(* LS Electric XG5000 project: V2H *)
(* PLC NewPLC *)
(* module base 0 slot 0: Input/Output Module:XEC-DR64H (DC 24V INPUT/RELAY OUTPUT, 64points) *)
(* module base 0 slot 1: Analog Input Module:XBF-AD04A (Volt/Current, 4-CH) *)
(* module base 0 slot 2: Analog IO Module:XBF-AH04A (I/O, 2/2 CH) *)
VAR_GLOBAL
    _01_CH0_ACT AT %UX0.1.16 : BOOL; (* Analog Input Module: CH0 Active *)
    _01_CH0_DATA AT %UW0.1.2 : WORD; (* Analog Input Module: CH0 Output *)
    _01_CH1_ACT AT %UX0.1.17 : BOOL; (* Analog Input Module: CH1 Active *)
    _01_CH1_DATA AT %UW0.1.3 : WORD; (* Analog Input Module: CH1 Output *)
    _01_CH2_ACT AT %UX0.1.18 : BOOL; (* Analog Input Module: CH2 Active *)
    _01_CH2_DATA AT %UW0.1.4 : WORD; (* Analog Input Module: CH2 Output *)
    _02_DA0_ACT AT %UX0.2.18 : BOOL; (* Analog IO Module: Output CH0 Active *)
    _02_DA0_OUTEN AT %UX0.2.96 : BOOL; (* Analog IO Module: Output CH0 Status Setting *)
    _02_DA1_DATA AT %UW0.2.8 : WORD; (* Analog IO Module: Output CH1 DATA *)
END_VAR

PROGRAM NewProgram_Copy (* task: Scan Program *)
VAR
    aa : REAL;
    AAAA : WORD;
    aaaaaaaaaaaaaaa : REAL;
    acCONTROL AT %IX0.0.0 : BOOL;
    ACTRANS : BOOL;
    ADD1 : WORD;
    ADD2 : WORD;
    AUTO AT %MX1 : BOOL;
    autoinhibit : BOOL;
    BLOCK : UINT;
    chillerready : BOOL;
    COMPRESSOR : BOOL;
    CONACTOR100 AT %IX0.0.21 : BOOL;
    CONTACTOR10 AT %IX0.0.3 : BOOL;
    CONTACTOR20 AT %IX0.0.4 : BOOL;
    CONTACTOR30 AT %IX0.0.8 : BOOL;
    CONTACTOR40 AT %IX0.0.9 : BOOL;
    CONTACTOR50 AT %IX0.0.10 : BOOL;
    CRITICALPRESSURE : BOOL;
    damperon : BOOL;
    damperramp : BOOL;
    DAMPERREF : WORD;
    DCPOWERK : BOOL;
    ddddddd : BOOL;
    DIRTYFILTER : BOOL;
    disk11kman : BOOL;
    disk1kman : BOOL;
    DIV11 : WORD;
    DIV12 : INT;
    DIV124 : INT;
    DIV2 : WORD;
    DIV21 : WORD;
    DIV22 : WORD;
    DIV23 : WORD;
    DIV32 : INT;
    DIV33 : INT;
    DP1SUBP1MACHIN : WORD;
    DP1SUBP1MACHIN2 : WORD;
    DP1SUBP1MACHININT : INT;
    DP2INT : INT;
    DP2RATE : INT;
    DPINT : INT;
    DPMUL : WORD;
    DPSUBZERO : INT;
    drive11kman : BOOL;
    DRIVE11KW AT %QX0.0.10 : BOOL;
    DRIVE75KW AT %QX0.0.9 : BOOL;
    DRIVEK1 AT %MX90 : BOOL;
    DRIVEK2 AT %MX91 : BOOL;
    DRIVEK3 : BOOL;
    DRIVEK4 : BOOL;
    DRIVEK5 : BOOL;
    DRIVEK6 : BOOL;
    DRIVEPUMP AT %MX92 : BOOL;
    dvi2 : DWORD;
    E1 : INT;
    E11 : REAL;
    E1REAL : REAL;
    E2 : WORD;
    EE : WORD;
    EE1 : WORD;
    EE2 : WORD;
    EMERGENCY AT %IX0.0.23 : BOOL;
    ERR : BOOL;
    ET : TIME;
    ET70 : TIME;
    fanon : BOOL;
    FANREFSCALE : WORD;
    FANRUN : BOOL;
    filterdisk : BOOL;
    filterjaroob : BOOL;
    FILTERMEDIA : BOOL;
    FILTERRUN : BOOL;
    FR1 AT %IX0.0.14 : BOOL;
    FR2 AT %IX0.0.15 : BOOL;
    FR3 AT %IX0.0.16 : BOOL;
    FR4 AT %IX0.0.17 : BOOL;
    FR5 AT %IX0.0.18 : BOOL;
    FR6 AT %IX0.0.19 : BOOL;
    GEARBOXK5 AT %QX0.0.5 : BOOL;
    gearboxman : BOOL;
    HIGHLIMDP : WORD;
    hihelimdpint : INT;
    HIMIDITYSCAL2 : WORD;
    HUMID2 : WORD;
    HUMID3 : WORD;
    HUMID4 : BOOL;
    HUMID5 : BOOL;
    HUMIDHIVALUE1 : WORD;
    HUMIDITIERR1 : WORD;
    HUMIDITYOUTSCAL : WORD;
    HUMIDLOWLIM1 : WORD;
    HUMIDNO1 : BOOL;
    HUMIDON : BOOL;
    hummidd : WORD;
    IN1 : SINT;
    IN10 : WORD;
    incin : WORD;
    inhumreal : REAL;
    inhumreal1 : REAL;
    inrealhuscale : REAL;
    inrealhuscale1 : REAL;
    INST : TON;
    INST1 : TON;
    INST10 : PIDRUN;
    INST11 : PIDRUN;
    INST12 : TON_UINT;
    INST13 : TON_UINT;
    INST14 : TON;
    INST15 : TON;
    INST16 : TON;
    INST17 : TON;
    INST18 : TON;
    INST19 : TON;
    INST2 : TON;
    INST20 : TON;
    INST21 : TON;
    INST22 : TON;
    INST23 : TON;
    INST24 : TON;
    INST25 : TON;
    INST26 : CTU_INT;
    INST27 : TON;
    INST28 : TON;
    INST29 : CTU_INT;
    INST3 : TON;
    INST30 : TON;
    INST31 : TON;
    INST32 : TON;
    INST33 : TON;
    INST34 : TON;
    INST35 : TON;
    INST36 : TON;
    INST37 : CTU_INT;
    INST38 : CTU_INT;
    INST39 : TON;
    INST4 : TON;
    INST40 : TON_UINT;
    INST41 : TON_UINT;
    INST42 : TON_UINT;
    INST43 : TON_UINT;
    INST44 : TON_UINT;
    INST45 : TON_UINT;
    INST46 : TON_UINT;
    INST47 : TMR;
    INST48 : TON_UINT;
    INST49 : TON_UINT;
    INST5 : TON;
    INST50 : TON_UINT;
    INST51 : TON_UINT;
    INST52 : TON_UINT;
    INST53 : TON;
    INST54 : TON;
    INST55 : TON;
    INST56 : TON;
    INST57 : TON;
    INST58 : TON;
    INST59 : TON;
    INST6 : TON;
    INST60 : TON;
    INST61 : TON;
    INST62 : TON;
    INST63 : TON;
    INST64 : TON;
    INST65 : TON;
    INST66 : TON_UINT;
    INST67 : TON;
    INST68 : TON;
    INST69 : TON;
    INST7 : TON;
    INST70 : TON_UINT;
    INST71 : TON;
    INST72 : TON;
    INST73 : TON;
    INST74 : TON;
    INST75 : TON;
    INST76 : TON;
    INST77 : TON_UINT;
    INST78 : TON_UINT;
    INST79 : TON;
    INST8 : TON;
    INST80 : TON;
    INST81 : TON;
    INST82 : TON;
    INST83 : TON;
    INST84 : TON;
    INST85 : TON;
    INST86 : TON;
    INST87 : TON;
    INST88 : TON;
    INST89 : TON;
    INST9 : TON;
    INST90 : TON_UINT;
    JAROOBK4 AT %QX0.0.4 : BOOL;
    jaroobman : BOOL;
    K1B AT %MX95 : BOOL;
    K2B AT %MX97 : BOOL;
    K2BYPASSDISK AT %QX0.0.2 : BOOL;
    K2DISK AT %QX0.0.1 : BOOL;
    K3B : BOOL;
    K3DISK1KW AT %QX0.0.3 : BOOL;
    K4B : BOOL;
    K5B : BOOL;
    K6B : BOOL;
    KBYPASS20 AT %IX0.0.5 : BOOL;
    KDISCH1 AT %MX96 : BOOL;
    KDISCH2 : BOOL;
    KDISCH3 : BOOL;
    KSUC AT %MX94 : BOOL;
    KSUC2 : BOOL;
    KSUC3 : BOOL;
    LASTDP2 : WORD;
    LOOP : UINT;
    man1 : BOOL;
    man10 : BOOL;
    man2 : BOOL;
    man3 : BOOL;
    man4 : BOOL;
    man5 : BOOL;
    man6 : BOOL;
    man7 : BOOL;
    man8 : BOOL;
    man9 : BOOL;
    meanfan : BOOL;
    meanfanman : BOOL;
    mesnfanman : BOOL;
    mot1 : BOOL;
    mot10 : BOOL;
    mot11 : BOOL;
    mot12 : BOOL;
    mot2 : BOOL;
    mot3 : BOOL;
    mot4 : BOOL;
    mot5 : BOOL;
    mot6 : BOOL;
    mot7 : BOOL;
    mot8 : BOOL;
    mot9 : BOOL;
    motor10 : BOOL;
    motor11 : BOOL;
    motor12 : BOOL;
    motor13 : BOOL;
    motor9 : BOOL;
    o1 : REAL;
    O10 : REAL;
    O11 : REAL;
    O13 : INT;
    O14 : INT;
    O2 : REAL;
    O3 : INT;
    ooot : INT;
    OUT : WORD;
    OUT10 : INT;
    OUT100 : INT;
    OUT101 : REAL;
    OUT102 : REAL;
    OUT103 : INT;
    OUT104 : WORD;
    OUT20 : INT;
    OUT200 : WORD;
    OUT202 : REAL;
    OUT205 : INT;
    OUT21 : INT;
    OUT300 : INT;
    OUT301 : REAL;
    OUT304 : INT;
    OUT305 : REAL;
    OUT306 : REAL;
    OUT308 : WORD;
    OUT314 : INT;
    OUT315 : REAL;
    OUT316 : REAL;
    OUT324 : INT;
    OUT325 : REAL;
    OUT326 : REAL;
    OUT330 : BOOL;
    out350 : BOOL;
    OUT400 : INT;
    OUT401 : REAL;
    OUT50 : WORD;
    OUT6 : WORD;
    OUT6bit : BOOL;
    outhumreal : REAL;
    OUTrealhuscale : REAL;
    OUTTMP : WORD;
    OUTTMPLOWLIM : WORD;
    ouuu : INT;
    ouuuuuuut : DWORD;
    P1MACHINSINT : INT;
    P2MAXINT : INT;
    P2MAXREAL : REAL;
    P2MININT : INT;
    PID_STAT : WORD;
    PTCSWITCH AT %IX0.0.20 : BOOL;
    PUMPON : BOOL;
    RESETTIMER : BOOL;
    rstauto : BOOL;
    RUNOK AT %MX98 : BOOL;
    scal11 : REAL;
    scale22 : REAL;
    scale23 : REAL;
    setauto AT %MX68 : BOOL;
    STATE1 : BOOL;
    STATE2 : BOOL;
    STATE3 : BOOL;
    STATE4 : BOOL;
    STATE5 : BOOL;
    STATE6 : BOOL;
    STATE7 : BOOL;
    step1 : BOOL;
    step10 : BOOL;
    step2 : BOOL;
    step3 : BOOL;
    step4 : BOOL;
    step5 : BOOL;
    step6 : BOOL;
    step7 : BOOL;
    step8 : BOOL;
    step9 : BOOL;
    SUBDP : WORD;
    SUCTION1RUN : BOOL;
    SUMMER : BOOL;
    teee : INT;
    TEMPE11 : INT;
    TEMPLOWLIM1 : WORD;
    TEMPLOWLIM2 : INT;
    TEMPMAX1 : WORD;
    TEMPMAX2 : INT;
    VFD1 : BOOL;
    VFD1FAULT AT %IX0.0.1 : BOOL;
    VFD1RUN AT %IX0.0.6 : BOOL;
    VFD2 : BOOL;
    VFD2FAULT AT %IX0.0.2 : BOOL;
    VFD2RUN AT %IX0.0.7 : BOOL;
    WINTER : BOOL;
END_VAR
VAR RETAIN
    DAMPERMAX AT %WW228 : INT;
    DAMPERMIN AT %WW230 : INT;
    DIV1 : WORD;
    DP AT %WW202 : WORD;
    DP1 AT %WW400 : WORD;
    DP2 AT %WW402 : INT;
    DP2SURGE AT %WW210 : INT;
    DP3 AT %WW404 : INT;
    FRMAX AT %WW224 : INT;
    FRMIN AT %WW226 : INT;
    INVERTERREF AT %WW500 : INT;
    P1MACHIN AT %WW200 : WORD;
    P2MAX AT %WW206 : WORD;
    P2MIN AT %WW208 : WORD;
    P3CRITICAL AT %WW218 : INT;
    P3MAX AT %WW214 : INT;
    P3MIN AT %WW216 : INT;
    scale1 AT %WD379 : REAL;
    scale2 AT %WD377 : REAL;
    SCALE21 AT %WD387 : REAL;
    Tacc AT %WW12 : WORD;
    TaccFan AT %WW204 : WORD;
    TFILTEROFF AT %WW222 : WORD;
    TFILTERON AT %WW220 : WORD;
    TSURGE AT %WW212 : WORD;
    VACUMEFRQ AT %WW232 : WORD;
    VIBRATION AT %WW234 : WORD;
END_VAR
VAR_EXTERNAL
    _01_CH0_ACT : BOOL; (* AT %UX0.1.16 *) (* Analog Input Module: CH0 Active *)
    _01_CH0_DATA : WORD; (* AT %UW0.1.2 *) (* Analog Input Module: CH0 Output *)
    _01_CH1_ACT : BOOL; (* AT %UX0.1.17 *) (* Analog Input Module: CH1 Active *)
    _01_CH1_DATA : WORD; (* AT %UW0.1.3 *) (* Analog Input Module: CH1 Output *)
    _01_CH2_ACT : BOOL; (* AT %UX0.1.18 *) (* Analog Input Module: CH2 Active *)
    _01_CH2_DATA : WORD; (* AT %UW0.1.4 *) (* Analog Input Module: CH2 Output *)
    _02_DA0_ACT : BOOL; (* AT %UX0.2.18 *) (* Analog IO Module: Output CH0 Active *)
    _02_DA0_OUTEN : BOOL; (* AT %UX0.2.96 *) (* Analog IO Module: Output CH0 Status Setting *)
    _02_DA1_DATA : WORD; (* AT %UW0.2.8 *) (* Analog IO Module: Output CH1 DATA *)
END_VAR
VAR
    _e1 : R_TRIG;
    _p2 : BOOL;
    _e3 : R_TRIG;
    _e4 : R_TRIG;
    _e5 : F_TRIG;
    _e6 : F_TRIG;
    _e7 : R_TRIG;
    _e8 : R_TRIG;
    _e9 : R_TRIG;
    _e10 : R_TRIG;
    _e11 : F_TRIG;
    _t12 : BOOL;
    _t13 : BOOL;
    _t14 : BOOL;
    _t15 : BOOL;
    _t16 : BOOL;
    _e17 : R_TRIG;
    _t18 : BOOL;
    _t19 : BOOL;
    _t20 : BOOL;
    _t21 : BOOL;
    _t22 : BOOL;
    _e23 : R_TRIG;
    _t24 : BOOL;
    _t25 : BOOL;
    _t26 : BOOL;
    _e27 : R_TRIG;
    _t28 : BOOL;
    _t29 : BOOL;
    _t30 : BOOL;
    _t31 : BOOL;
END_VAR

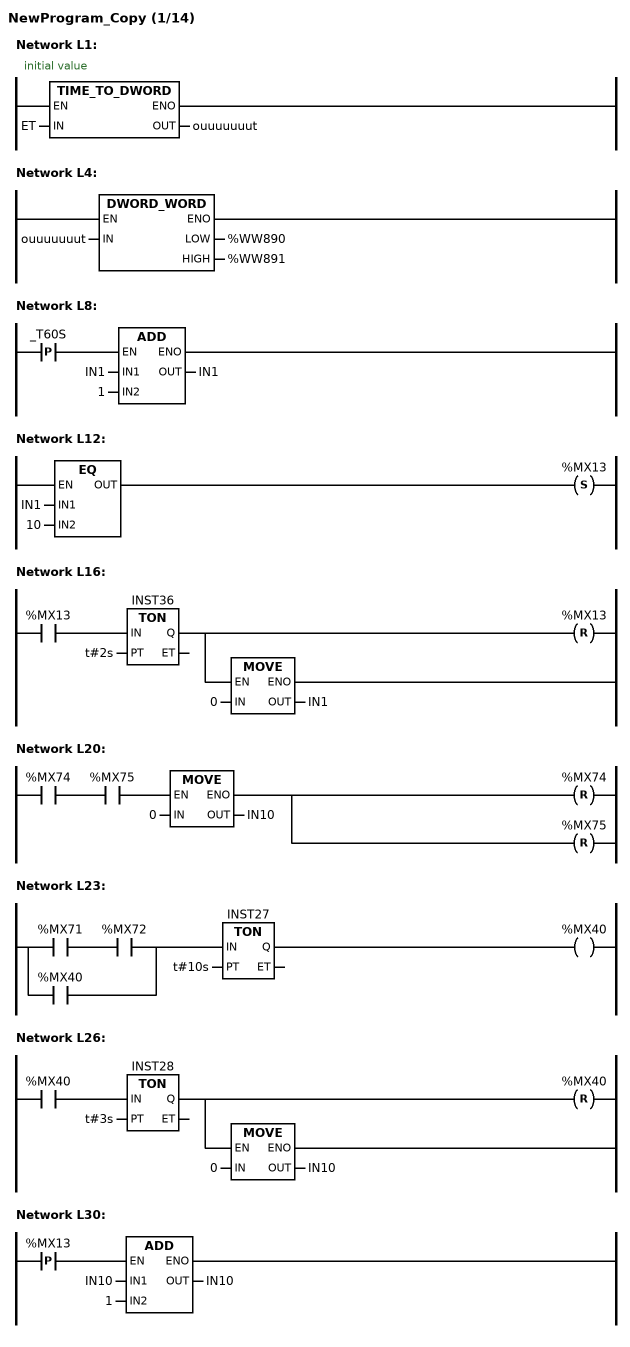
(* initial value *)
(* Rung L1 *)
ouuuuuuut := TIME_TO_DWORD(ET);
(* Rung L4 *)
%WW890 := DWORD_WORD(IN := ouuuuuuut, HIGH => %WW891);
(* Rung L8 *)
_e1(CLK := _T60S);
IF _e1.Q THEN IN1 := IN1 + 1; END_IF;
(* Rung L12 *)
IF IN1 = 10 THEN %MX13 := TRUE; END_IF;
(* Rung L16 *)
INST36(IN := %MX13, PT := t#2s);
IF INST36.Q THEN
    %MX13 := FALSE;
    IN1 := 0;
END_IF;
(* Rung L20 *)
IF %MX74 AND %MX75 THEN IN10 := 0; END_IF;
_p2 := %MX74 AND %MX75;
IF _p2 THEN
    %MX74 := FALSE;
    %MX75 := FALSE;
END_IF;
(* Rung L23 *)
INST27(IN := (%MX71 AND %MX72) OR %MX40, PT := t#10s);
%MX40 := INST27.Q;
(* Rung L26 *)
INST28(IN := %MX40, PT := t#3s);
IF INST28.Q THEN
    %MX40 := FALSE;
    IN10 := 0;
END_IF;
(* Rung L30 *)
_e3(CLK := %MX13);
IF _e3.Q THEN IN10 := IN10 + 1; END_IF;

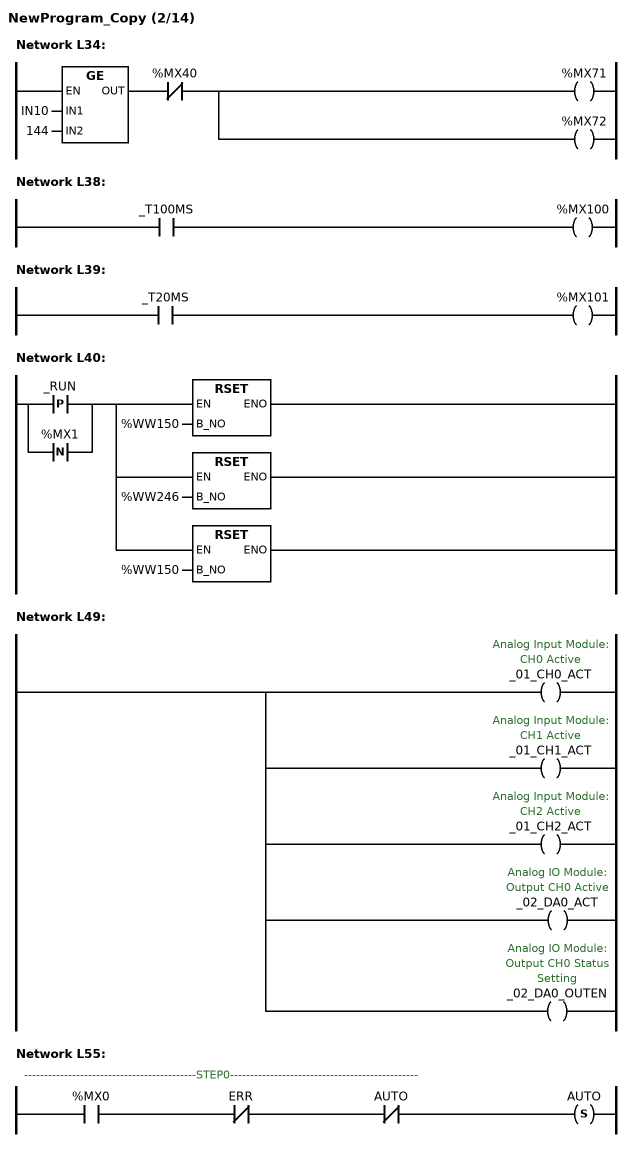
(* Rung L34 *)
%MX71 := (IN10 >= 144) AND NOT %MX40;
%MX72 := (IN10 >= 144) AND NOT %MX40;
(* Rung L38 *)
%MX100 := _T100MS;
(* Rung L39 *)
%MX101 := _T20MS;
(* Rung L40 *)
_e4(CLK := _RUN);
_e5(CLK := %MX1);
IF _e4.Q OR _e5.Q THEN
    RSET(B_NO := %WW150);
    RSET(B_NO := %WW246);
    RSET(B_NO := %WW150);
END_IF;
(* Rung L49 *)
_01_CH0_ACT := TRUE;
_01_CH1_ACT := TRUE;
_01_CH2_ACT := TRUE;
_02_DA0_ACT := TRUE;
_02_DA0_OUTEN := TRUE;
(* -------------------------------------------STEP0----------------------------------------------- *)
(* Rung L55 *)
IF %MX0 AND NOT ERR AND NOT AUTO THEN AUTO := TRUE; END_IF;

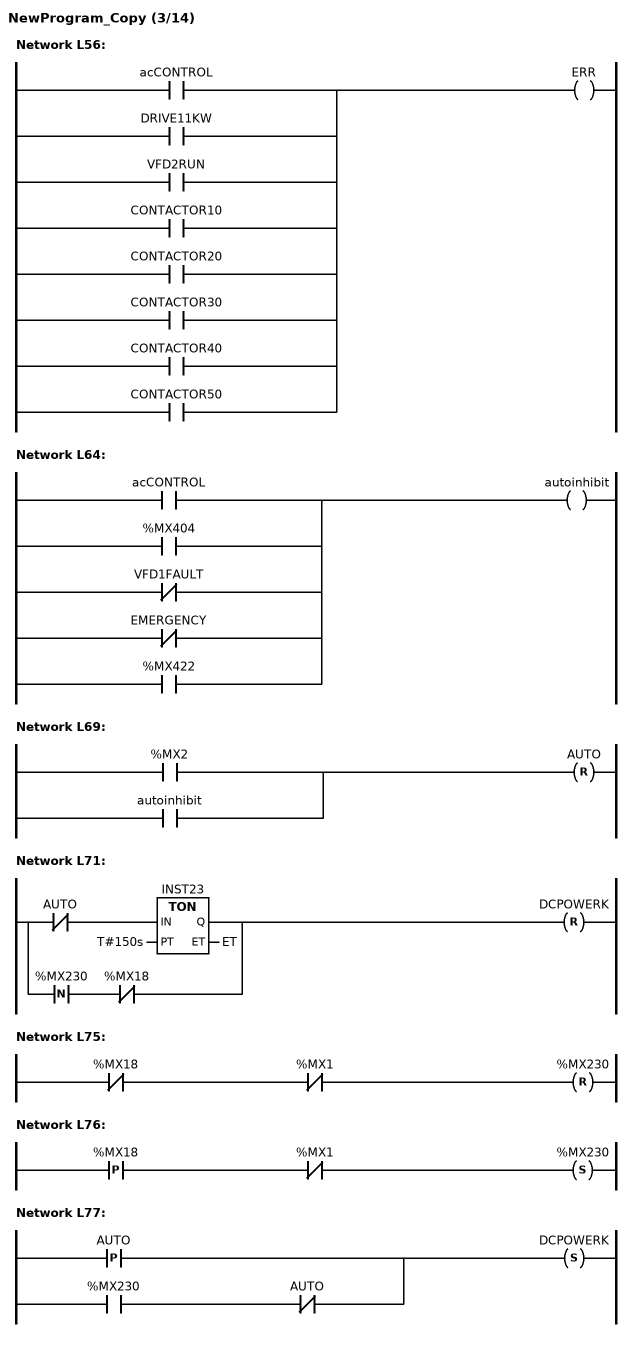
(* Rung L56 *)
ERR := acCONTROL OR DRIVE11KW OR VFD2RUN OR CONTACTOR10 OR CONTACTOR20 OR CONTACTOR30 OR CONTACTOR40 OR CONTACTOR50;
(* Rung L64 *)
autoinhibit := acCONTROL OR %MX404 OR NOT VFD1FAULT OR NOT EMERGENCY OR %MX422;
(* Rung L69 *)
IF %MX2 OR autoinhibit THEN AUTO := FALSE; END_IF;
(* Rung L71 *)
INST23(IN := NOT AUTO, PT := T#150s, ET => ET);
_e6(CLK := %MX230);
IF INST23.Q OR (_e6.Q AND NOT %MX18) THEN DCPOWERK := FALSE; END_IF;
(* Rung L75 *)
IF NOT %MX18 AND NOT %MX1 THEN %MX230 := FALSE; END_IF;
(* Rung L76 *)
_e7(CLK := %MX18);
IF _e7.Q AND NOT %MX1 THEN %MX230 := TRUE; END_IF;
(* Rung L77 *)
_e8(CLK := AUTO);
IF _e8.Q OR (%MX230 AND NOT AUTO) THEN DCPOWERK := TRUE; END_IF;

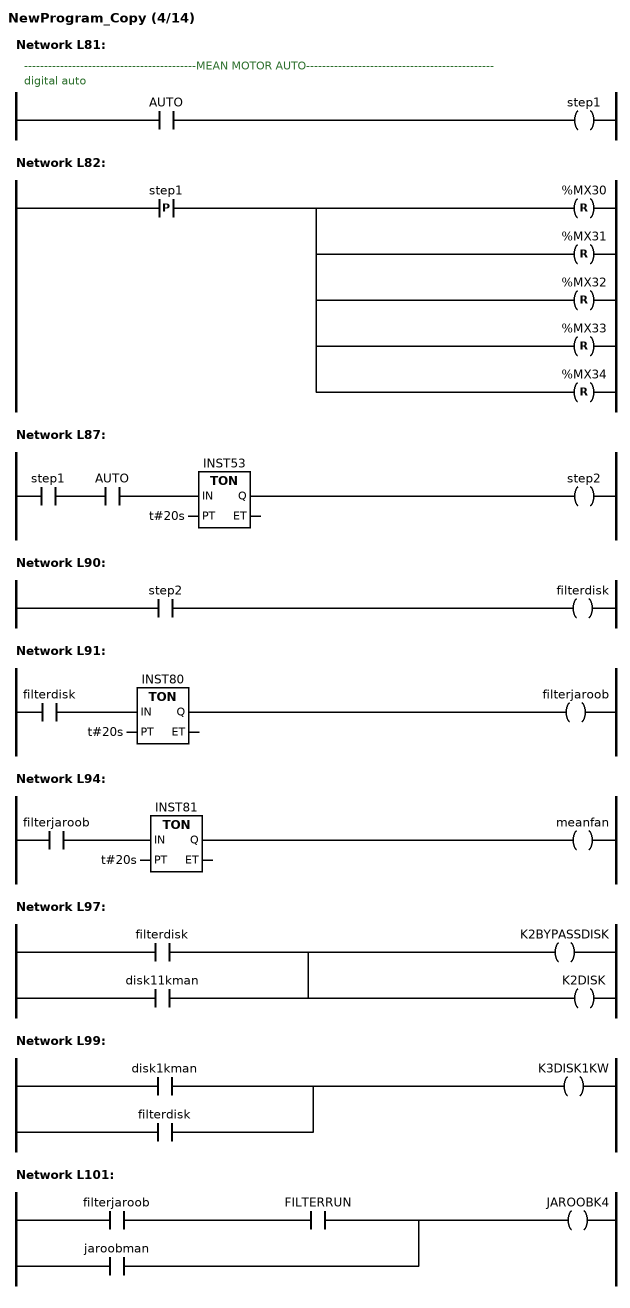
(* -------------------------------------------MEAN MOTOR AUTO----------------------------------------------- *)
(* digital auto *)
(* Rung L81 *)
step1 := AUTO;
(* Rung L82 *)
_e9(CLK := step1);
IF _e9.Q THEN
    %MX30 := FALSE;
    %MX31 := FALSE;
    %MX32 := FALSE;
    %MX33 := FALSE;
    %MX34 := FALSE;
END_IF;
(* Rung L87 *)
INST53(IN := step1 AND AUTO, PT := t#20s);
step2 := INST53.Q;
(* Rung L90 *)
filterdisk := step2;
(* Rung L91 *)
INST80(IN := filterdisk, PT := t#20s);
filterjaroob := INST80.Q;
(* Rung L94 *)
INST81(IN := filterjaroob, PT := t#20s);
meanfan := INST81.Q;
(* Rung L97 *)
K2BYPASSDISK := filterdisk OR disk11kman;
K2DISK := filterdisk OR disk11kman;
(* Rung L99 *)
K3DISK1KW := disk1kman OR filterdisk;
(* Rung L101 *)
JAROOBK4 := (filterjaroob AND FILTERRUN) OR jaroobman;

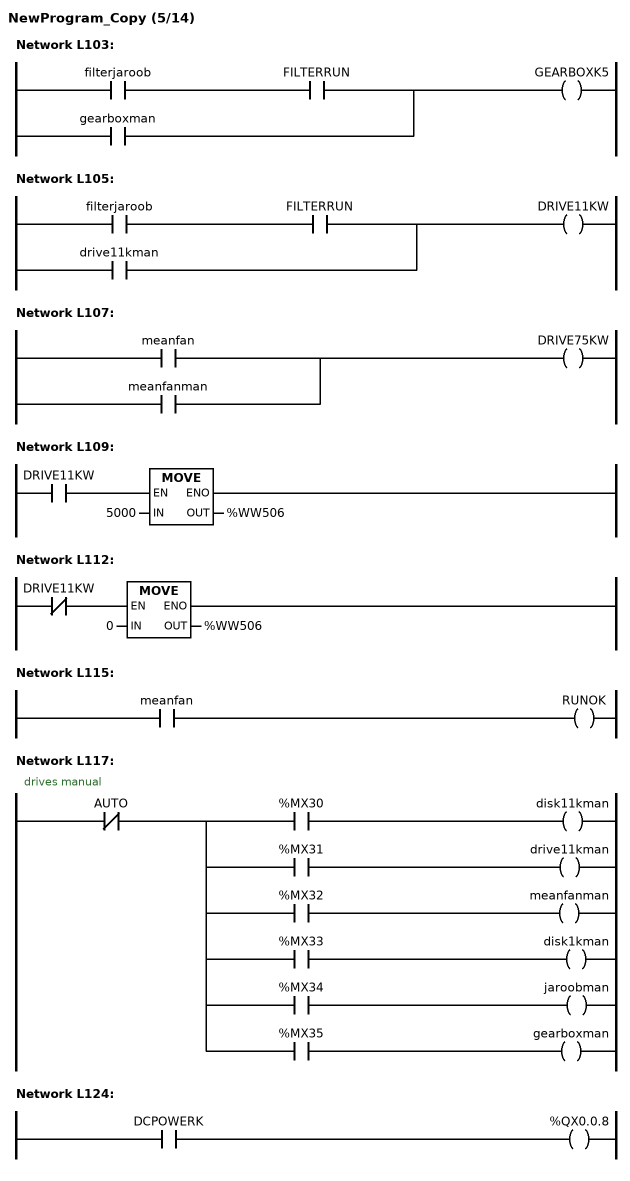
(* Rung L103 *)
GEARBOXK5 := (filterjaroob AND FILTERRUN) OR gearboxman;
(* Rung L105 *)
DRIVE11KW := (filterjaroob AND FILTERRUN) OR drive11kman;
(* Rung L107 *)
DRIVE75KW := meanfan OR meanfanman;
(* Rung L109 *)
IF DRIVE11KW THEN %WW506 := 5000; END_IF;
(* Rung L112 *)
IF NOT DRIVE11KW THEN %WW506 := 0; END_IF;
(* Rung L115 *)
RUNOK := meanfan;
(* drives manual *)
(* Rung L117 *)
disk11kman := NOT AUTO AND %MX30;
drive11kman := NOT AUTO AND %MX31;
meanfanman := NOT AUTO AND %MX32;
disk1kman := NOT AUTO AND %MX33;
jaroobman := NOT AUTO AND %MX34;
gearboxman := NOT AUTO AND %MX35;
(* Rung L124 *)
%QX0.0.8 := DCPOWERK;

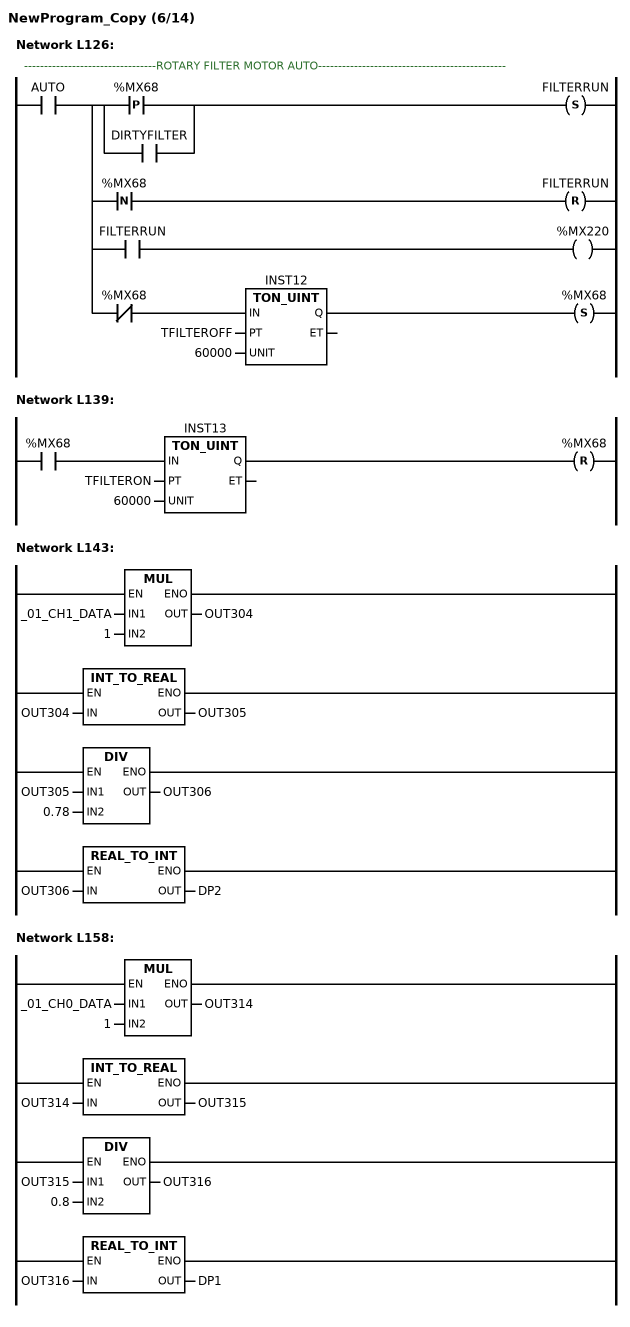
(* ---------------------------------ROTARY FILTER MOTOR AUTO----------------------------------------------- *)
(* Rung L126 *)
_e10(CLK := %MX68);
IF AUTO AND (_e10.Q OR DIRTYFILTER) THEN FILTERRUN := TRUE; END_IF;
_e11(CLK := %MX68);
IF AUTO AND _e11.Q THEN FILTERRUN := FALSE; END_IF;
%MX220 := AUTO AND FILTERRUN;
INST12(IN := AUTO AND NOT %MX68, PT := TFILTEROFF, UNIT := 60000);
IF INST12.Q THEN %MX68 := TRUE; END_IF;
(* Rung L139 *)
INST13(IN := %MX68, PT := TFILTERON, UNIT := 60000);
IF INST13.Q THEN %MX68 := FALSE; END_IF;
(* Rung L143 *)
OUT304 := _01_CH1_DATA * 1;
OUT305 := INT_TO_REAL(OUT304);
OUT306 := OUT305 / 0.78;
DP2 := REAL_TO_INT(OUT306);
(* Rung L158 *)
OUT314 := _01_CH0_DATA * 1;
OUT315 := INT_TO_REAL(OUT314);
OUT316 := OUT315 / 0.8;
DP1 := REAL_TO_INT(OUT316);

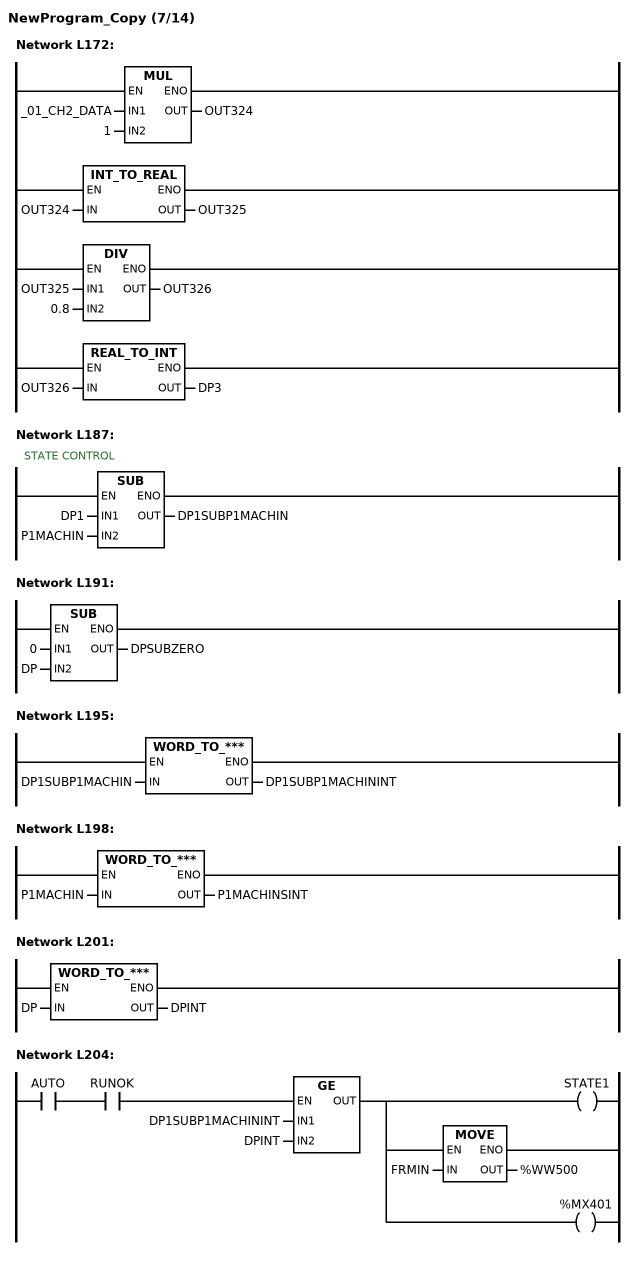
(* Rung L172 *)
OUT324 := _01_CH2_DATA * 1;
OUT325 := INT_TO_REAL(OUT324);
OUT326 := OUT325 / 0.8;
DP3 := REAL_TO_INT(OUT326);
(* STATE CONTROL *)
(* Rung L187 *)
DP1SUBP1MACHIN := DP1 - P1MACHIN;
(* Rung L191 *)
DPSUBZERO := 0 - DP;
(* Rung L195 *)
DP1SUBP1MACHININT := WORD_TO_***(DP1SUBP1MACHIN);
(* Rung L198 *)
P1MACHINSINT := WORD_TO_***(P1MACHIN);
(* Rung L201 *)
DPINT := WORD_TO_***(DP);
(* Rung L204 *)
IF AUTO AND RUNOK THEN _t12 := DP1SUBP1MACHININT >= DPINT; END_IF;
STATE1 := _t12;
IF _t12 THEN %WW500 := FRMIN; END_IF;
%MX401 := _t12;

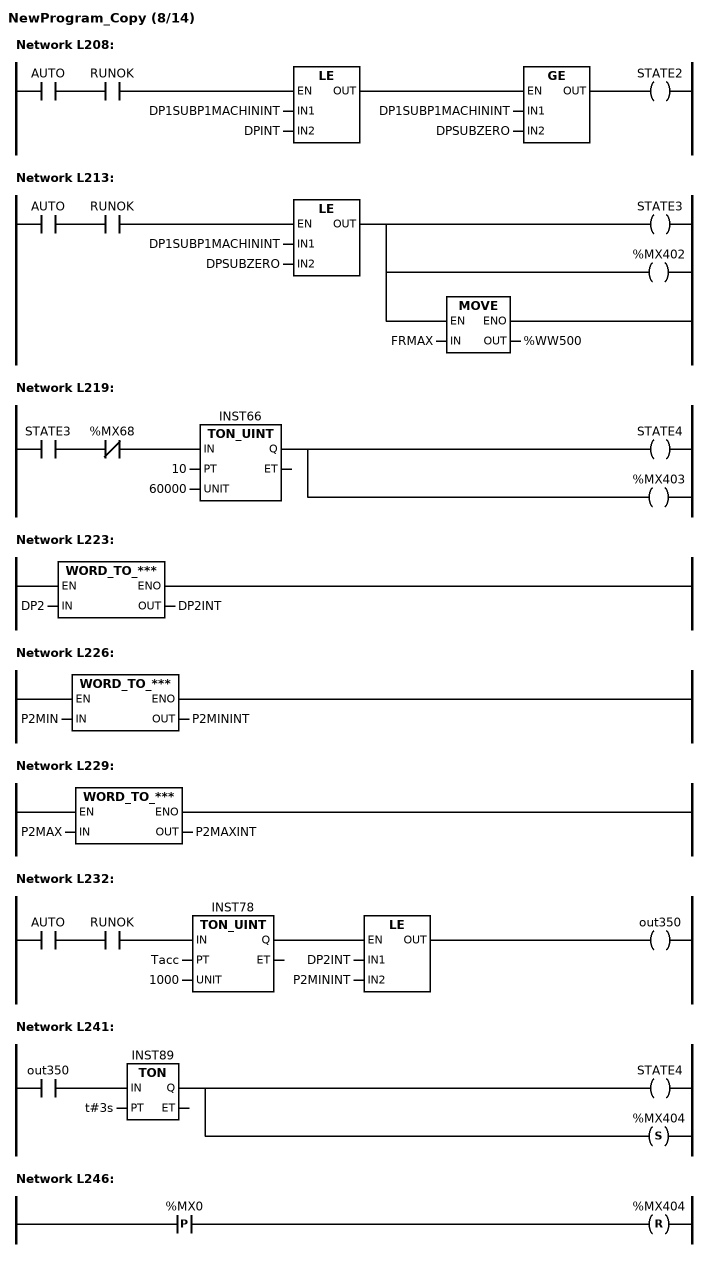
(* Rung L208 *)
IF AUTO AND RUNOK THEN _t13 := DP1SUBP1MACHININT <= DPINT; END_IF;
IF _t13 THEN _t14 := DP1SUBP1MACHININT >= DPSUBZERO; END_IF;
STATE2 := _t14;
(* Rung L213 *)
IF AUTO AND RUNOK THEN _t15 := DP1SUBP1MACHININT <= DPSUBZERO; END_IF;
STATE3 := _t15;
%MX402 := _t15;
IF _t15 THEN %WW500 := FRMAX; END_IF;
(* Rung L219 *)
INST66(IN := STATE3 AND NOT %MX68, PT := 10, UNIT := 60000);
STATE4 := INST66.Q;
%MX403 := INST66.Q;
(* Rung L223 *)
DP2INT := WORD_TO_***(DP2);
(* Rung L226 *)
P2MININT := WORD_TO_***(P2MIN);
(* Rung L229 *)
P2MAXINT := WORD_TO_***(P2MAX);
(* Rung L232 *)
INST78(IN := AUTO AND RUNOK, PT := Tacc, UNIT := 1000);
IF INST78.Q THEN _t16 := DP2INT <= P2MININT; END_IF;
out350 := _t16;
(* Rung L241 *)
INST89(IN := out350, PT := t#3s);
STATE4 := INST89.Q;
IF INST89.Q THEN %MX404 := TRUE; END_IF;
(* Rung L246 *)
_e17(CLK := %MX0);
IF _e17.Q THEN %MX404 := FALSE; END_IF;

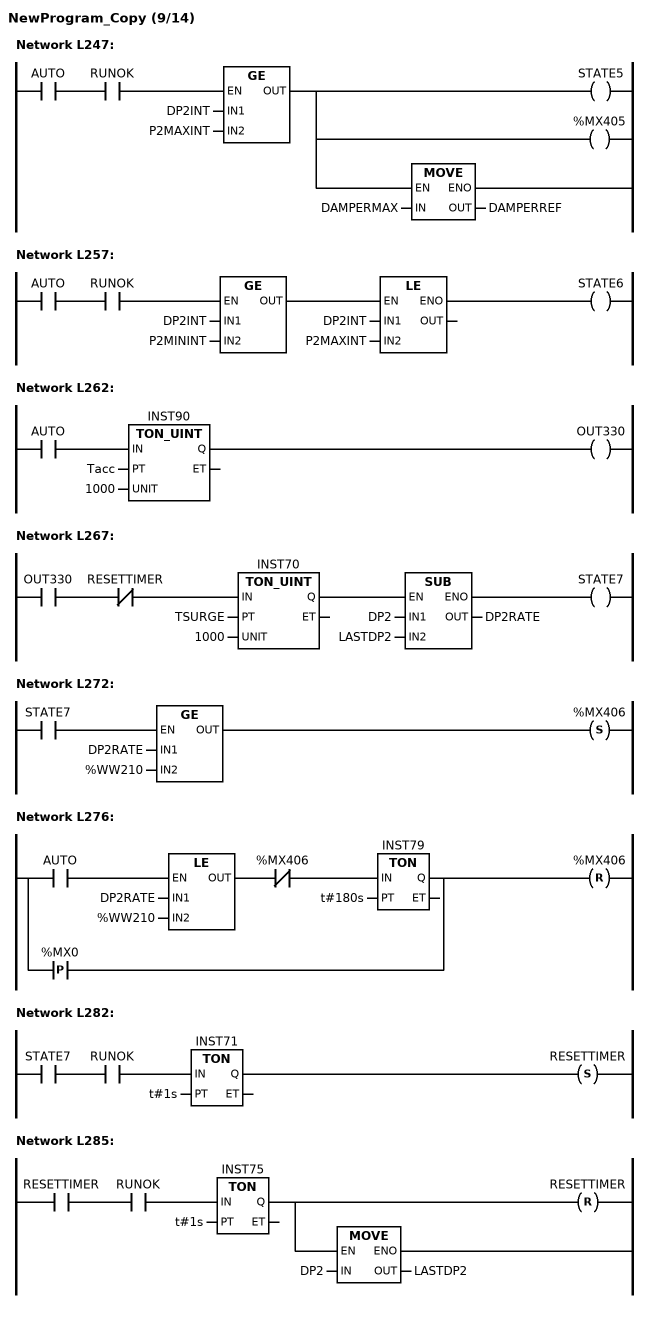
(* Rung L247 *)
IF AUTO AND RUNOK THEN _t18 := DP2INT >= P2MAXINT; END_IF;
STATE5 := _t18;
%MX405 := _t18;
IF _t18 THEN DAMPERREF := DAMPERMAX; END_IF;
(* Rung L257 *)
IF AUTO AND RUNOK THEN _t19 := DP2INT >= P2MININT; END_IF;
IF _t19 THEN _t20 := DP2INT <= P2MAXINT; END_IF;
STATE6 := _t19;
(* Rung L262 *)
INST90(IN := AUTO, PT := Tacc, UNIT := 1000);
OUT330 := INST90.Q;
(* Rung L267 *)
INST70(IN := OUT330 AND NOT RESETTIMER, PT := TSURGE, UNIT := 1000);
IF INST70.Q THEN DP2RATE := DP2 - LASTDP2; END_IF;
STATE7 := INST70.Q;
(* Rung L272 *)
IF STATE7 THEN _t21 := DP2RATE >= %WW210; END_IF;
IF _t21 THEN %MX406 := TRUE; END_IF;
(* Rung L276 *)
IF AUTO THEN _t22 := DP2RATE <= %WW210; END_IF;
INST79(IN := _t22 AND NOT %MX406, PT := t#180s);
_e23(CLK := %MX0);
IF INST79.Q OR _e23.Q THEN %MX406 := FALSE; END_IF;
(* Rung L282 *)
INST71(IN := STATE7 AND RUNOK, PT := t#1s);
IF INST71.Q THEN RESETTIMER := TRUE; END_IF;
(* Rung L285 *)
INST75(IN := RESETTIMER AND RUNOK, PT := t#1s);
IF INST75.Q THEN
    RESETTIMER := FALSE;
    LASTDP2 := DP2;
END_IF;

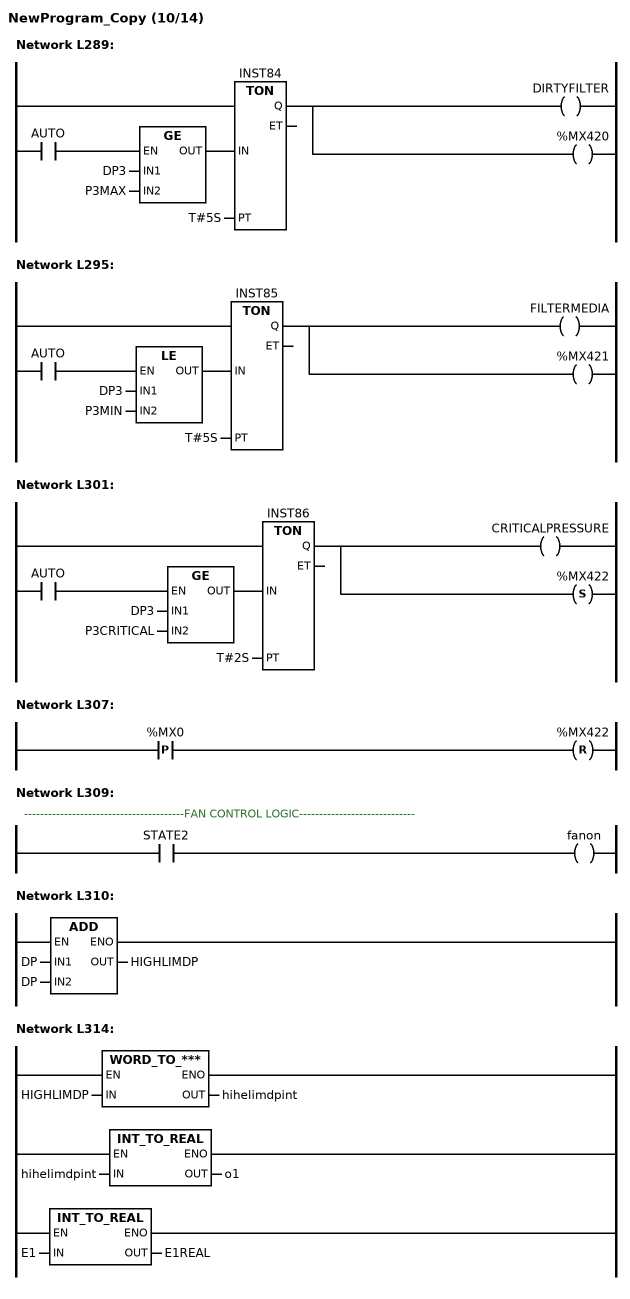
(* Rung L289 *)
IF AUTO THEN _t24 := DP3 >= P3MAX; END_IF;
INST84(IN := _t24, PT := T#5S);
DIRTYFILTER := INST84.Q;
%MX420 := INST84.Q;
(* Rung L295 *)
IF AUTO THEN _t25 := DP3 <= P3MIN; END_IF;
INST85(IN := _t25, PT := T#5S);
FILTERMEDIA := INST85.Q;
%MX421 := INST85.Q;
(* Rung L301 *)
IF AUTO THEN _t26 := DP3 >= P3CRITICAL; END_IF;
INST86(IN := _t26, PT := T#2S);
CRITICALPRESSURE := INST86.Q;
IF INST86.Q THEN %MX422 := TRUE; END_IF;
(* Rung L307 *)
_e27(CLK := %MX0);
IF _e27.Q THEN %MX422 := FALSE; END_IF;
(* ----------------------------------------FAN CONTROL LOGIC----------------------------- *)
(* Rung L309 *)
fanon := STATE2;
(* Rung L310 *)
HIGHLIMDP := DP + DP;
(* Rung L314 *)
hihelimdpint := WORD_TO_***(HIGHLIMDP);
o1 := INT_TO_REAL(hihelimdpint);
E1REAL := INT_TO_REAL(E1);

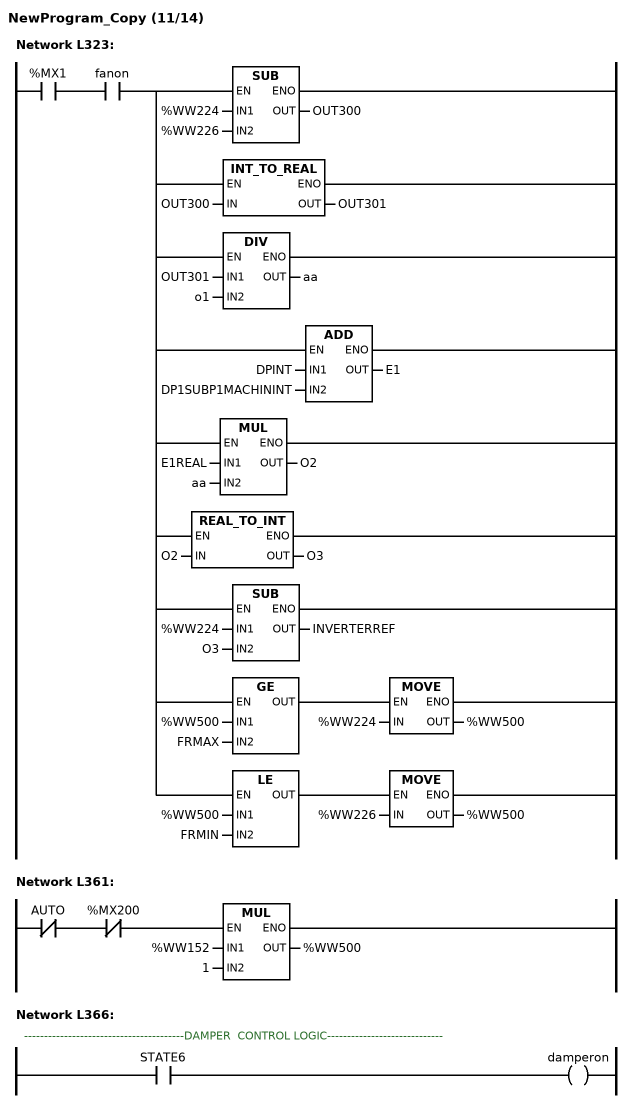
(* Rung L323 *)
IF %MX1 AND fanon THEN
    OUT300 := %WW224 - %WW226;
    OUT301 := INT_TO_REAL(OUT300);
    aa := OUT301 / o1;
    E1 := DPINT + DP1SUBP1MACHININT;
    O2 := E1REAL * aa;
    O3 := REAL_TO_INT(O2);
    INVERTERREF := %WW224 - O3;
    _t28 := %WW500 >= FRMAX;
END_IF;
IF _t28 THEN %WW500 := %WW224; END_IF;
IF %MX1 AND fanon THEN _t29 := %WW500 <= FRMIN; END_IF;
IF _t29 THEN %WW500 := %WW226; END_IF;
(* Rung L361 *)
IF NOT AUTO AND NOT %MX200 THEN %WW500 := %WW152 * 1; END_IF;
(* ----------------------------------------DAMPER  CONTROL LOGIC----------------------------- *)
(* Rung L366 *)
damperon := STATE6;

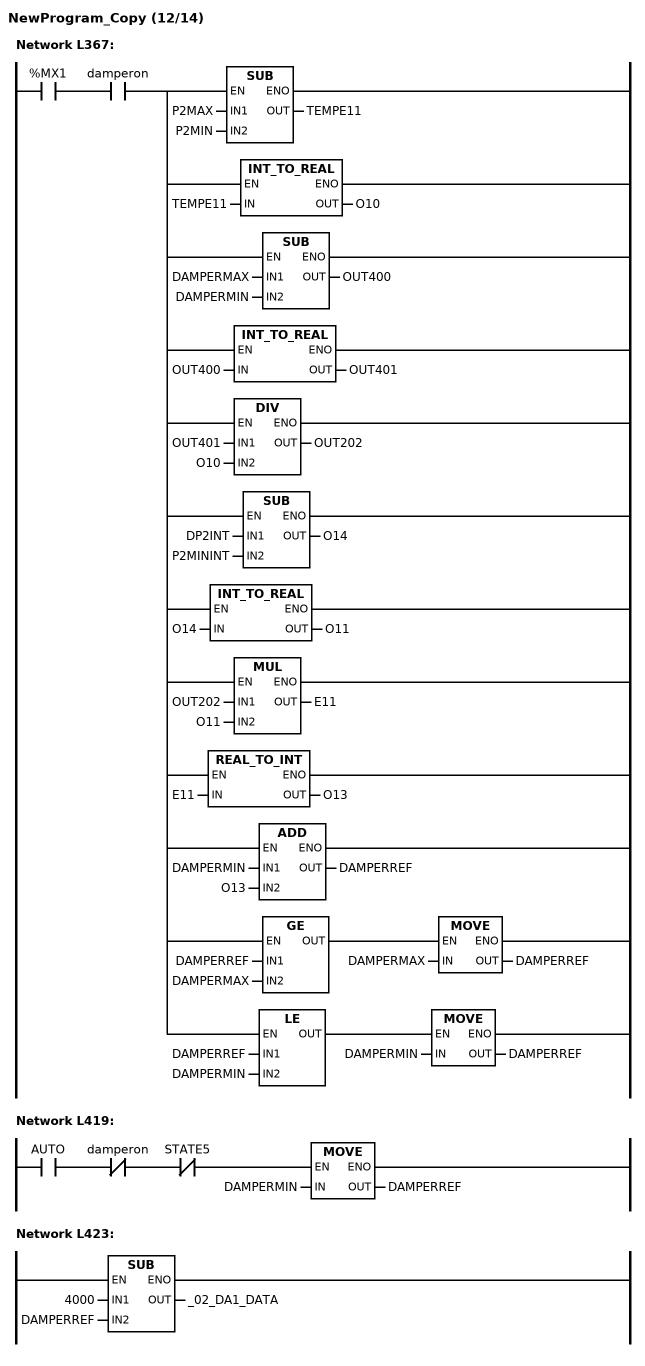
(* Rung L367 *)
IF %MX1 AND damperon THEN
    TEMPE11 := P2MAX - P2MIN;
    O10 := INT_TO_REAL(TEMPE11);
    OUT400 := DAMPERMAX - DAMPERMIN;
    OUT401 := INT_TO_REAL(OUT400);
    OUT202 := OUT401 / O10;
    O14 := DP2INT - P2MININT;
    O11 := INT_TO_REAL(O14);
    E11 := OUT202 * O11;
    O13 := REAL_TO_INT(E11);
    DAMPERREF := DAMPERMIN + O13;
    _t30 := DAMPERREF >= DAMPERMAX;
END_IF;
IF _t30 THEN DAMPERREF := DAMPERMAX; END_IF;
IF %MX1 AND damperon THEN _t31 := DAMPERREF <= DAMPERMIN; END_IF;
IF _t31 THEN DAMPERREF := DAMPERMIN; END_IF;
(* Rung L419 *)
IF AUTO AND NOT damperon AND NOT STATE5 THEN DAMPERREF := DAMPERMIN; END_IF;
(* Rung L423 *)
_02_DA1_DATA := 4000 - DAMPERREF;

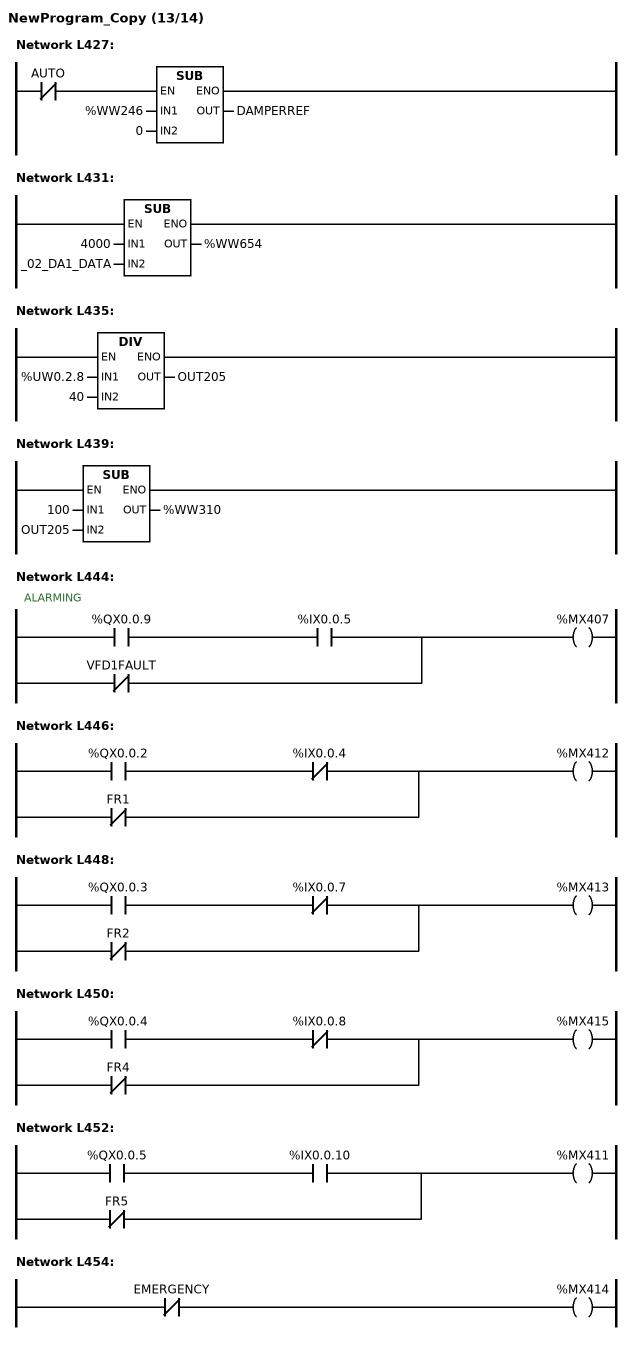
(* Rung L427 *)
IF NOT AUTO THEN DAMPERREF := %WW246 - 0; END_IF;
(* Rung L431 *)
%WW654 := 4000 - _02_DA1_DATA;
(* Rung L435 *)
OUT205 := %UW0.2.8 / 40;
(* Rung L439 *)
%WW310 := 100 - OUT205;
(* ALARMING *)
(* Rung L444 *)
%MX407 := (%QX0.0.9 AND %IX0.0.5) OR NOT VFD1FAULT;
(* Rung L446 *)
%MX412 := (%QX0.0.2 AND NOT %IX0.0.4) OR NOT FR1;
(* Rung L448 *)
%MX413 := (%QX0.0.3 AND NOT %IX0.0.7) OR NOT FR2;
(* Rung L450 *)
%MX415 := (%QX0.0.4 AND NOT %IX0.0.8) OR NOT FR4;
(* Rung L452 *)
%MX411 := (%QX0.0.5 AND %IX0.0.10) OR NOT FR5;
(* Rung L454 *)
%MX414 := NOT EMERGENCY;

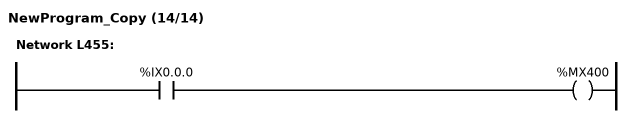
(* Rung L455 *)
%MX400 := %IX0.0.0;
END_PROGRAM